TYPE
	jog_manager_command_enum: (
	JOG_MANAGER_CMD_NONE						:= 0,	(*$ No command assigned $*)
	JOG_MANAGER_SET_ACTIVATION_CONDITION		:= 1,
	JOG_MANAGER_RESET_ACTIVATION_CONDITION		:= 2,
	JOG_MANAGER_STOP_ABSOLUTE_MOVEMENT			:= 3
	) := JOG_MANAGER_CMD_NONE;
END_TYPE

(* stored: Version 1.1.0.1, ProductVersion 3.1.4022.12
   DUT jog_manager_command_enum: Id {35e801e7-2069-49ed-9882-719d14ae7b83} *)
